FUNCTION_BLOCK T_SubModuleMock IMPLEMENTS I_PackML_BaseModule
VAR_INPUT
	dontInitialise : BOOL;
	_error : BOOL;
END_VAR
VAR_OUTPUT
	_newState	: Tc3_PackML_V2.E_PMLCommand;
	_newMode : E_PMLUnitMode;
	_initComplete, cyclicHasBeenCalled : BOOL;
END_VAR

{warning 'add property implementation'}
PROPERTY Busy : BOOL
GET
END_GET
END_PROPERTY

METHOD ChangeMode
VAR_INPUT
	Mode	: E_PMLUnitMode;
END_VAR
_newMode := Mode;
END_METHOD

METHOD ChangeState
VAR_INPUT
	State	: Tc3_PackML_V2.E_PMLCommand;
END_VAR
_newState := State;
END_METHOD

{warning 'add property implementation'}
PROPERTY CurrentAlarmSeverity : TcEventSeverity
GET
END_GET
END_PROPERTY

{warning 'add property implementation'}
PROPERTY CurrentMode : E_PMLUnitMode
GET
END_GET
END_PROPERTY

{warning 'add property implementation'}
PROPERTY CurrentState : Tc3_PackML_V2.E_PMLState
GET
END_GET
END_PROPERTY

METHOD CyclicLogic
cyclicHasBeenCalled := TRUE;

IF NOT dontInitialise THEN
	_initComplete := TRUE;
END_IF
END_METHOD

{warning 'add property implementation'}
PROPERTY Error : BOOL
GET
Error := _error;
END_GET
END_PROPERTY

{warning 'add property implementation'}
PROPERTY ErrorID : UDINT
GET
END_GET
END_PROPERTY

{warning 'add property implementation'}
PROPERTY InitComplete : BOOL
GET
InitComplete := _initComplete;
END_GET
END_PROPERTY

{warning 'add property implementation'}
PROPERTY LogModeChanges : BOOL
GET
END_GET
SET
END_SET
END_PROPERTY

{warning 'add property implementation'}
PROPERTY LogStateChanges : BOOL
GET
END_GET
SET
END_SET
END_PROPERTY

{warning 'add property implementation'}
PROPERTY ModeCommand : DINT
GET
END_GET
SET
END_SET
END_PROPERTY

{warning 'add property implementation'}
PROPERTY Name : STRING
GET
END_GET
SET
END_SET
END_PROPERTY

{warning 'add property implementation'}
PROPERTY ParentResponseDefinitions : ARRAY [0..4] OF SPT_BaseTypes.E_AlarmResponse
GET
END_GET
SET
END_SET
END_PROPERTY

{warning 'add property implementation'}
PROPERTY StateCommand : Tc3_PackML_V2.E_PMLCommand
GET
END_GET
SET
END_SET
END_PROPERTY

END_FUNCTION_BLOCK

(* stored: Version 1.1.0.1, ProductVersion 3.1.4024.12
   POU T_SubModuleMock: Id {8d712bd5-9ca6-48bf-aba8-799ed79c3cc0}, SpecialFunc None
   Property Busy: Id {b9d941b2-8da1-47d1-8afe-bc8e40f0ad87}
   Get Get: Id {de3abd4b-219c-49f0-9bf0-7c70ef2ae43b}
   Method ChangeMode: Id {d3d7d6e2-2a84-480b-8703-08b512640cb7}
   Method ChangeState: Id {06ce365a-f76a-4bcc-adaa-ed5e694bf825}
   Property CurrentAlarmSeverity: Id {60fccc78-73da-44dd-95b6-b09c8fdb361b}
   Get Get: Id {9ed6efc8-aaff-4d06-b5a9-a02cf1116593}
   Property CurrentMode: Id {fd19641f-7de6-4733-8b93-5fa00b5c87da}
   Get Get: Id {1b7d5d42-6754-4582-9a7e-5d3ad6ec984c}
   Property CurrentState: Id {3acfc985-6d6a-4792-b605-c86a96b133bc}
   Get Get: Id {37191b55-2a91-4786-b540-345a0eb9c695}
   Method CyclicLogic: Id {1ff9707e-f47e-4191-9e00-5dc629f08ee5}
   Property Error: Id {d30e9e89-06e8-44c5-a2cd-523b0b18f25b}
   Get Get: Id {5fe3d98a-baea-4512-a61c-653ebb65ea6b}
   Property ErrorID: Id {75594b7f-8773-42c6-b299-82177ed1194a}
   Get Get: Id {fafdbd10-13dd-4819-8f0b-9a081232bc0a}
   Property InitComplete: Id {5c79abb6-c428-4925-a1e5-5215cd3d22b7}
   Get Get: Id {d39d9739-65fe-42b1-8638-a88760980564}
   Property LogModeChanges: Id {7fe55808-9cc7-45cb-8b8b-6ba2fa2603c4}
   Get Get: Id {608c4487-12f7-42d6-b1b7-a034f683ac2b}
   Set Set: Id {27e345d4-7804-43d5-8a8e-7435eecb528c}
   Property LogStateChanges: Id {4b5768b6-1e11-46a0-a737-e2e0d77b61a5}
   Get Get: Id {39e424f5-b80f-4dbe-92d7-4246e1fed0b6}
   Set Set: Id {88efdd6f-2018-4cd2-bf0f-92ae1ef201c9}
   Property ModeCommand: Id {af5844a4-da01-4f35-afbf-b9ddffa51189}
   Get Get: Id {a1f91e73-0966-4624-a67a-5651daaf5846}
   Set Set: Id {28bde9f9-dbe7-4a05-9d98-531924018830}
   Property Name: Id {e4d445f7-28b3-4b48-86e7-392f6dd65e41}
   Get Get: Id {64cc32ec-8aef-4b70-be14-9e375497ce27}
   Set Set: Id {355975df-7a4d-4afb-be78-989832bf828a}
   Property ParentResponseDefinitions: Id {c5e601f0-c85f-4526-b373-83bf80e7ed81}
   Get Get: Id {63120bb2-c3aa-4e4d-877a-85d16b227637}
   Set Set: Id {37948d72-77e3-424b-bd60-c6becbe362c0}
   Property StateCommand: Id {c883b793-b2a7-4d6e-99da-504e07cd660e}
   Get Get: Id {d00358a3-7c1e-47d1-819c-e885e23b9bd1}
   Set Set: Id {5684fb0a-8217-40f6-89ce-02a9947fe3b9} *)
